// TIA Portal V17 export
// export: Created 2022-07-28T18:02:51.1068585Z, ExportSetting None, DisplayName Totally Integrated Automation Portal, DisplayVersion V17, DisplayName TIA Portal Openness, DisplayVersion V17, DisplayName TIA Portal Teamcenter Gateway, DisplayVersion V17, DisplayName TIA Portal Version Control Interface, DisplayVersion V17, DisplayName TIA Portal Test Suite Advanced, DisplayVersion V17, DisplayName SINAMICS Startdrive Advanced, DisplayVersion V17, DisplayName SINAMICS DCC, DisplayVersion V17, DisplayName SINAMICS Startdrive G130, G150, S120, S150, SINAMICS MV, S210, DisplayVersion V17, DisplayName SINAMICS Startdrive G110M, G120, G120C, G120D, G120P, G115D, DisplayVersion V17, DisplayName STEP 7 Professional, DisplayVersion V17, DisplayName SIMATIC Energy Suite, DisplayVersion V17, DisplayName STEP 7 CFC, DisplayVersion V17, DisplayName STEP 7 Safety, DisplayVersion V17, DisplayName WinCC Advanced / Unified PC, DisplayVersion V17, DisplayName SIMATIC Visualization Architect, DisplayVersion V17
FUNCTION_BLOCK "Lib_FB_SlideGate_Blow"   // FB63, SCL
{ S7_Optimized_Access := 'TRUE' }
// stored: AutoNumber false, MemoryReserve 100, SetENOAutomatically false
   VAR_INPUT
      I_Initialization { ExternalAccessible := 'False'; ExternalVisible := 'False'; ExternalWritable := 'False'} : Bool := FALSE;   // 1 = Restart PLC is active (First scan)
      IR_CycleTime { ExternalAccessible := 'False'; ExternalVisible := 'False'; ExternalWritable := 'False'} : Real := 0.0;   // Time of last PLC cycle, sec
      II_Obj_ID { ExternalAccessible := 'False'; ExternalVisible := 'False'; ExternalWritable := 'False'} : Int := -1;   // Tech ID of object
      I_CmdGeneralReset { ExternalAccessible := 'False'; ExternalVisible := 'False'; ExternalWritable := 'False'} : Bool;   // 0 ⮥ 1 = Input general reset ERROR/Interlocks
      I_One_1s { ExternalAccessible := 'False'; ExternalVisible := 'False'; ExternalWritable := 'False'} : Bool;   // 1 = One cycle per one seccond pulse
      I_EstopHMI { ExternalAccessible := 'False'; ExternalVisible := 'False'; ExternalWritable := 'False'} : Bool := TRUE;   // 0 = HMI/WinCC Emergency stop active
      I_SuppyBox_Ok { ExternalAccessible := 'False'; ExternalVisible := 'False'; ExternalWritable := 'False'} : Bool := TRUE;   // 1 = Release from supply box where exist object
      I_IsOpen { ExternalAccessible := 'False'; ExternalVisible := 'False'; ExternalWritable := 'False'} : Bool;   // Repeat status of opened sensor
      I_IsClose { ExternalAccessible := 'False'; ExternalVisible := 'False'; ExternalWritable := 'False'} : Bool;   // Repeat status of closed sensor
      I_GenFaultMainDrive { ExternalAccessible := 'False'; ExternalVisible := 'False'; ExternalWritable := 'False'} : Bool := TRUE;   // 1 = ППП/Гібридкий контактор/ПЧ в нормі// 0 = Аварія
      I_CmdAutoFromInputFB { ExternalAccessible := 'False'; ExternalVisible := 'False'; ExternalWritable := 'False'} : Bool;   // 1 = Команди AutoMode беруться із входу FB // 0 = Команди AutoMode беруться із масиву AutoArray
      I_CmdAutoOpen { ExternalAccessible := 'False'; ExternalVisible := 'False'; ExternalWritable := 'False'} : Bool;   // (if IB_CmdAutoFromInputFB==1) 1 = In auto mode the motor to run in open direction until the open interlock becomes false, or this input is set low"
      I_CmdAutoClose { ExternalAccessible := 'False'; ExternalVisible := 'False'; ExternalWritable := 'False'} : Bool;   // (if IB_CmdAutoFromInputFB==1) 1 = In auto mode the motor to run in close direction until the close interlock becomes false, or this input is set low"
      I_ManLocalModeActive { ExternalAccessible := 'False'; ExternalVisible := 'False'; ExternalWritable := 'False'} : Bool;   // Switching in external mode ManualLocal if PRM.ManLocalPirority=1(hight)
      I_CmdManLocalOpen { ExternalAccessible := 'False'; ExternalVisible := 'False'; ExternalWritable := 'False'} : Bool;   // 1 = In ManualLocal mode the motor to run in open direction until the open interlock becomes false, or this input is set low
      I_CmdManLocalClose { ExternalAccessible := 'False'; ExternalVisible := 'False'; ExternalWritable := 'False'} : Bool;   // 1 = In ManualLocal mode the motor to run in close direction until the close interlock becomes false, or this input is set low
      IB_InterlocksOpen_8 { ExternalAccessible := 'False'; ExternalVisible := 'False'; ExternalWritable := 'False'} : Byte;   // <>0 = Interlock active - One or more from 8 Interlocks active // 1bit <--> 1 Interlock
      IB_InterlocksClose_8 { ExternalAccessible := 'False'; ExternalVisible := 'False'; ExternalWritable := 'False'} : Byte;   // <>0 = Interlock active - One or more from 8 Interlocks active // 1bit <--> 1 Interlock
      IW_ExternalError_16 { ExternalAccessible := 'False'; ExternalVisible := 'False'; ExternalWritable := 'False'} : Word;   // <>0 = External error active - One or more from 16 error active // 1bit <--> 1 error
      I_ExternalWarning { ExternalAccessible := 'False'; ExternalVisible := 'False'; ExternalWritable := 'False'} : Bool;   // 1 = External Warning
   END_VAR
   VAR_OUTPUT
      Q_CmdOpen { ExternalAccessible := 'False'; ExternalVisible := 'False'; ExternalWritable := 'False'} : Bool;   // 1 = Motor commanded open /Activation output / State transferred to physical output
      Q_IsOpen { ExternalAccessible := 'False'; ExternalVisible := 'False'; ExternalWritable := 'False'} : Bool;   // Repeat status of opened sensor
      Q_IsClose { ExternalAccessible := 'False'; ExternalVisible := 'False'; ExternalWritable := 'False'} : Bool;   // Repeat status of closed sensor
      Q_Reset { ExternalAccessible := 'False'; ExternalVisible := 'False'; ExternalWritable := 'False'} : Bool;   // 1 = Reset faults
      Q_Error { ExternalAccessible := 'False'; ExternalVisible := 'False'; ExternalWritable := 'False'} : Bool;   // This output indicates whether theres an error/fault condition in the motor
      Q_Warning { ExternalAccessible := 'False'; ExternalVisible := 'False'; ExternalWritable := 'False'} : Bool;   // This output indicates whether theres an warning condition in the motor
      Q_Auto { ExternalAccessible := 'False'; ExternalVisible := 'False'; ExternalWritable := 'False'} : Bool;   // 1= Automatic operating mode active
      Q_ManLocal { ExternalAccessible := 'False'; ExternalVisible := 'False'; ExternalWritable := 'False'} : Bool;   // 1= ManualLocal operating mode active
      Q_Stoped { ExternalAccessible := 'False'; ExternalVisible := 'False'; ExternalWritable := 'False'} : Bool;   // 1= Motor Stoped
      Q_Run { ExternalAccessible := 'False'; ExternalVisible := 'False'; ExternalWritable := 'False'} : Bool;   // 1= Motor running
      Q_RunOpen { ExternalAccessible := 'False'; ExternalVisible := 'False'; ExternalWritable := 'False'} : Bool;   // 1= Motor running open
      Q_RunClose { ExternalAccessible := 'False'; ExternalVisible := 'False'; ExternalWritable := 'False'} : Bool;   // 1= Motor running close
      Q_DataErr { ExternalAccessible := 'False'; ExternalVisible := 'False'; ExternalWritable := 'False'} : Bool;   // 1 = Transfer data error occured (ObjDB -> temp, ect)
   END_VAR
   VAR_IN_OUT
      IQ_PLC_CycleInfo : Variant;   // Ref to data about PLC cycle
   END_VAR
   VAR
      s_RequestOpen { ExternalAccessible := 'False'; ExternalVisible := 'False'; ExternalWritable := 'False'} : Bool;   // 1 = Request for start in Open dirrection for all modes
      s_TON_Plausible { ExternalAccessible := 'False'; ExternalVisible := 'False'; ExternalWritable := 'False'} : "Lib_FB_Timer_ON_Simple";
      s_TON_Pause { ExternalAccessible := 'False'; ExternalVisible := 'False'; ExternalWritable := 'False'} : "Lib_FB_Timer_ON_Simple";
      s_TP_Work { ExternalAccessible := 'False'; ExternalVisible := 'False'; ExternalWritable := 'False'} : "Lib_FB_Timer_TP_Simple";
      s_EdgeAuto { ExternalAccessible := 'False'; ExternalVisible := 'False'; ExternalWritable := 'False'} : "Lib_FB_Edge";
      s_EdgeActivOpen { ExternalAccessible := 'False'; ExternalVisible := 'False'; ExternalWritable := 'False'} : "Lib_FB_Edge";
      s_EdgeActivClose { ExternalAccessible := 'False'; ExternalVisible := 'False'; ExternalWritable := 'False'} : "Lib_FB_Edge";
      s_EdgeSim { ExternalAccessible := 'False'; ExternalVisible := 'False'; ExternalWritable := 'False'} : "Lib_FB_Edge";
      s_EdgeLocal { ExternalAccessible := 'False'; ExternalVisible := 'False'; ExternalWritable := 'False'} : "Lib_FB_Edge";
      s_EdgeError { ExternalAccessible := 'False'; ExternalVisible := 'False'; ExternalWritable := 'False'} : "Lib_FB_Edge";
      s_EdgeWarning { ExternalAccessible := 'False'; ExternalVisible := 'False'; ExternalWritable := 'False'} : "Lib_FB_Edge";
   END_VAR
   VAR RETAIN
      s_Simulation { ExternalAccessible := 'False'; ExternalVisible := 'False'; ExternalWritable := 'False'} : Struct   // Data for simulation process
         Obj_DATA_BACKUP : Struct   // MOTOR NORMAL MODE DATA BACKUP FOR SIMULATION MODE
            Config : "_SlideGate_Blow_Config";
            Counters : "_SlideGate_Blow_Counters";
            sud_MotoHours_Electro : "_MotoHours_One";
            sud_MotoHours_Mech : "_MotoHours_One";
         END_STRUCT;
      END_STRUCT;
      s_Obj_Retain_BUp { ExternalAccessible := 'False'; ExternalVisible := 'False'; ExternalWritable := 'False'} : Struct
         Config : "_SlideGate_Blow_Config";
         Counters : "_SlideGate_Blow_Counters";
         Mode : "UDT_Mode";
      END_STRUCT;
   END_VAR
   VAR
      s_TP_ResetOut { ExternalAccessible := 'False'; ExternalVisible := 'False'; ExternalWritable := 'False'} : "Lib_FB_Timer_TP_Simple";
   END_VAR
   VAR_TEMP
      t_DataErr : Bool;   // 1 = Transfer data error occured (ObjDB -> temp, ect)
      t_PlausibleCondition : Bool;   // 1 = Conition for detect plausible error
      t_ReleaseStart : Bool;   // 1 = Release for start in any mode
      t_RequestActive : Bool;   // 1 = Request is active for any mode in any dirrection
      t_RequestOpenActive : Bool;   // 1 = Request is active for any mode in Open dirrection
      t_RequestCloseActive : Bool;   // 1 = Request is active for any mode in Close dirrection
      t_ResetLogic : Bool;   // 1 = Reset all signals for logic
      ti_CMDLogic : Int;   // Command word for logic
      tui_NumObjDB : UInt;   // Number of DB for storage object data
      tui_MaxObjects : UInt;   // Max number of objects in plant
      tui_DB_ShiftHMI : UInt;   // Object DB number shift
      tui_DB_ShiftPLC : UInt;   // Object DB number shift
      tui_DBSens_ShiftHMI : UInt;   // Object DB number shift
      tui_DBSens_ShiftPLC : UInt;   // Object DB number shift
      t_ObjAny_HMI : DB_ANY;   // Ref to object data
      t_ObjVar_HMI : Variant;   // Ref to object data
      t_ObjAny_PLC : DB_ANY;   // Ref to object data
      t_ObjVar_PLC : Variant;   // Ref to object data
      t_PB_HMI : Struct   // Buttons from HMI
         ResetError : Bool;   // + set-->CMD_ALMACK_tag -Reset errors pushbutton
         ManRunOpen : Bool;   // - Move Open in manual mode pushbutton
         ManRunClose : Bool;   // - Move Close in manual mode pushbutton
         ResetGeneralReset : Bool;   // -Reset Error + Interlock
         CntResetALL : Bool;   // - обнулити всі лічильники - (Total+Last+Alm+Wrn+)
         CntResetTimeTOT : Bool;   // - обнулити лічильник мотогодин (Total+Last)
         CntResetActTOT : Bool;   // - обнулити запусків (Total+Last)
         spare7 : Bool;
         spare8 : Bool;
         spare9 : Bool;
         spare10 : Bool;
         spare11 : Bool;
         spare12 : Bool;
         spare13 : Bool;
         spare14 : Bool;
         spare15 : Bool;
         spare16 : Bool;
         spare17 : Bool;
         spare18 : Bool;
         spare19 : Bool;
         spare20 : Bool;
         spare21 : Bool;
         spare22 : Bool;
         spare23 : Bool;
         spare24 : Bool;
         spare25 : Bool;
         spare26 : Bool;
         spare27 : Bool;
         spare28 : Bool;
         spare29 : Bool;
         spare30 : Bool;
         spare31 : Bool;
      END_STRUCT;
      t_Obj_HMI : "Lib_UDT_SlideGate_Blow_HMI";   // Object data
      t_Obj_PLC : "Lib_UDT_SlideGate_Blow_PLC";
      t_PLC_CycleInfo : "Lib_PLC_CycleInfo";   // Data about PLC cycle
      t_AutoControl : "Lib_UDT_AutoControl";   // Data for auto control module for current element
      t_InternalData : "Lib_UDT_Int";   // Internal data
      t_AutoControl_CMD : Struct   // Commands from auto control module for current element
         CmdAutoOpen : Bool;
         CmdAutoClose : Bool;
         CmdAutoOpenRaw : Bool;
         CmdAutoCloseRaw : Bool;
      END_STRUCT;
      t_Buffer : Array[0..100] of Byte;   // Buffer for use serialize
   END_VAR
   VAR CONSTANT
      cr_TimePlausible : Real := 5.0;   // Time for detectplausible error, s
      cr_TimeAddWalkErr : Real := 20.0;   // Additional time for walk error after autocalibrate, %
   END_VAR
BEGIN

   REGION Initialization/read data from out DB
       //Set internal data
       "Lib_FC_GenMoto_InitInternal"(#t_InternalData);

       //Reinit gen data
       #t_DataErr := false;
       #t_Obj_HMI.Config.w_enableExternalErrors_16 := w#16#FFFF;
       #t_Obj_HMI.Config.b_bypassInterlocksForward_8 := b#16#ff;
       #t_Obj_HMI.Config.b_bypassInterlocksReverse_8 := b#16#ff;
       #tui_MaxObjects := "D_General_ProgramDATA".ui_MaxObjects;
       #tui_DB_ShiftHMI := "D_General_ProgramDATA".ui_Shift_DB_HMI;
       #tui_DB_ShiftPLC := "D_General_ProgramDATA".ui_Shift_DB_PLC;
       #tui_DBSens_ShiftHMI := "D_General_ProgramDATA".ui_Shift_DBSens_HMI;
       #tui_DBSens_ShiftPLC := "D_General_ProgramDATA".ui_Shift_DBSens_PLC;
       //Read data PLC
       VariantGet(SRC := #IQ_PLC_CycleInfo,
                  DST => #t_PLC_CycleInfo);

       //Read Object data
       //Reinit temp values
       #t_Obj_HMI := "D_ZeroTypes".SlideGate_Blow_HMI;
       #t_Obj_PLC := "D_ZeroTypes".SlideGate_Blow_PLC;

       IF #II_Obj_ID >= 0
       THEN
           //Read HMI data
           #tui_NumObjDB := INT_TO_UINT(#II_Obj_ID) + #tui_DB_ShiftHMI;
           #t_ObjAny_HMI := UINT_TO_DB_ANY(#tui_NumObjDB);
           #t_ObjVar_HMI := DB_ANY_TO_VARIANT(in := #t_ObjAny_HMI, err => #t_InternalData.i_Tmp);

           //If DB exist and convertion without error
           IF #t_InternalData.i_Tmp = 0
           THEN
               VariantGet(SRC := #t_ObjVar_HMI,
                          DST => #t_Obj_HMI);
           ELSE
               #t_DataErr := true;
           END_IF;

           //Read PLC data
           #tui_NumObjDB := INT_TO_UINT(#II_Obj_ID) + #tui_DB_ShiftPLC;
           #t_ObjAny_PLC := UINT_TO_DB_ANY(#tui_NumObjDB);
           #t_ObjVar_PLC := DB_ANY_TO_VARIANT(in := #t_ObjAny_PLC, err => #t_InternalData.i_Tmp);

           //If DB exist and convertion without error
           IF #t_InternalData.i_Tmp = 0
           THEN
               VariantGet(SRC := #t_ObjVar_PLC,
                          DST => #t_Obj_PLC);
           ELSE
               #t_DataErr := true;
           END_IF;

       ELSE
           #t_DataErr := true;
       END_IF;

       //Read general info data
       #t_AutoControl := "DB_AutoControl_arr".AutoControl_arr[#tui_MaxObjects];
       CASE #II_Obj_ID OF
           0..999:  // ID of element in range
               #t_AutoControl := "DB_AutoControl_arr".AutoControl_arr[#II_Obj_ID];
           ELSE
               ;
       END_CASE;

       //Read retain data if initialization is active
       IF #I_Initialization
       THEN
           #t_Obj_HMI.Config := #s_Obj_Retain_BUp.Config;
           #t_Obj_HMI.Counters := #s_Obj_Retain_BUp.Counters;
           #t_Obj_PLC.Mode := #s_Obj_Retain_BUp.Mode;
       END_IF;
   END_REGION
   //---------------------------------------------------------------
   //---------------------------------------------------------------
   REGION Define CMD for block logic 
       //Reinit logic CMD
       #ti_CMDLogic := 0;

       //Define CMD by priority modes
       "Lib_FC_GenMoto_ChoiceCMD"(I_Mode := #t_Obj_PLC.Mode,
                                  QI_CMD_Logic => #ti_CMDLogic,
                                  IQI_CMD_Global := #t_PLC_CycleInfo.CMD_GLOBAL,
                                  IQI_CMD_Auto := #t_AutoControl.Global_CMD,
                                  IQI_CMD_HMI := #t_Obj_HMI.i_CMD);
   END_REGION
   //---------------------------------------------------------------
   //---------------------------------------------------------------
   REGION Switch modes  
       "Lib_FC_GenMoto_SwitchMode"(I_ManLocalModeActive := #I_ManLocalModeActive,
                                   IQI_CMD_Logic := #ti_CMDLogic,
                                   IQ_Mode := #t_Obj_PLC.Mode,
                                   IQ_ObjDataConfig := #t_Obj_HMI.Config,
                                   IQ_BUpDataConfig := #s_Simulation.Obj_DATA_BACKUP.Config,
                                   IQ_ObjDataCounters := #t_Obj_HMI.Counters,
                                   IQ_BUpDataCounters := #s_Simulation.Obj_DATA_BACKUP.Counters);

       #s_EdgeAuto(IB_Initialisation:=#I_Initialization,
                   IB_Input:=#t_Obj_PLC.Mode.Auto);
       #s_EdgeSim(IB_Initialisation:=#I_Initialization,
                  IB_Input:=#t_Obj_PLC.Mode.Simulation);
       #s_EdgeLocal(IB_Initialisation:=#I_Initialization,
                    IB_Input:=#t_Obj_PLC.Mode.ManualLocal);

   END_REGION
   //---------------------------------------------------------------
   //---------------------------------------------------------------
   REGION Commands & release for start in auto mode
       //Raw command for start in auto mode
       //-------------------------------------
       IF #I_CmdAutoFromInputFB
       THEN // Auto CMD from FB INPUT
           #t_AutoControl_CMD.CmdAutoOpenRaw := #I_CmdAutoOpen
           AND #t_Obj_PLC.Mode.Auto;
           #t_AutoControl_CMD.CmdAutoCloseRaw := #I_CmdAutoClose
           AND #t_Obj_PLC.Mode.Auto;

       ELSE // Auto CMD from AutoControl_array DB

           IF #t_Obj_PLC.Mode.Auto
           THEN
               IF #s_TP_Work.QB_TimerOut
               THEN
                   #t_AutoControl.CTW.%W0 := W#16#1;
                   #t_AutoControl.StatusGen.Release := true;
               ELSE
                   #t_AutoControl.CTW.%W0 := W#16#0;
                   #t_AutoControl.StatusGen.Release := false;
               END_IF;
           ELSE
               #t_AutoControl.CTW := dW#16#0;
               #t_AutoControl.StatusGen.Release := false;
           END_IF;

           #t_AutoControl_CMD.CmdAutoOpenRaw := (WORD_TO_UINT(#t_AutoControl.CTW.%W0) > 0)
           AND #t_AutoControl.StatusGen.Release;
           #t_AutoControl_CMD.CmdAutoCloseRaw := (WORD_TO_UINT(#t_AutoControl.CTW.%W1) > 0)
           AND #t_AutoControl.StatusGen.Release;

       END_IF;
       //-------------------------------------
       //-------------------------------------
       //Processed auto mode commands
       #t_AutoControl_CMD.CmdAutoOpen := #t_AutoControl_CMD.CmdAutoOpenRaw;
       #t_AutoControl_CMD.CmdAutoClose := #t_AutoControl_CMD.CmdAutoCloseRaw;

       REGION Timers for work and pause 
           #s_TON_Pause(IR_CycleTime:=#IR_CycleTime,
                        IB_StartTimerInput:=NOT #s_TP_Work.QB_TimerOut,
                        IB_ResetTimer:=NOT #t_Obj_PLC.Mode.Auto
                        OR NOT #t_Obj_PLC.State.Ready,
                        IR_SpTime:=#t_Obj_HMI.Config.r_SP_TimePause);

           #s_TP_Work(IR_CycleTime:=#IR_CycleTime,
                      IB_StartTimerInput:=#s_TON_Pause.QB_TimerOut
                      OR #s_EdgeAuto.QB_EdgePos,
                      IB_ResetTimer:=NOT #t_Obj_PLC.Mode.Auto
                      OR NOT #t_Obj_PLC.State.Ready,
                      IR_SpTime:=#t_Obj_HMI.Config.r_SP_TimeWork);

           //Left time
           IF #t_Obj_PLC.Mode.Auto
           THEN
               IF #s_TON_Pause.sR_Cv_ToDone > 0.0
               THEN
                   #t_Obj_HMI.Config.r_PV_LeftTime := #s_TON_Pause.sR_Cv_ToDone;
               ELSE
                   #t_Obj_HMI.Config.r_PV_LeftTime := 0.0;
               END_IF;
           ELSE
               #t_Obj_HMI.Config.r_PV_LeftTime := 0.0;
           END_IF;
       END_REGION


       //Reset release bit
      // #t_AutoControl.StatusGen.Release := false; 
   END_REGION
   //---------------------------------------------------------------
   //---------------------------------------------------------------
   REGION Convert commands to bit
       //Reinit all bits
       SCATTER(IN := #t_InternalData.d_Alw0,
               OUT => #t_PB_HMI);

       //Read commands and set apropriate bits
       CASE #ti_CMDLogic OF
           12:  // Start open in manual mode
               #t_PB_HMI.ManRunOpen := true;
           13:  // Start close in manual mode
               #t_PB_HMI.ManRunClose := true;
           19: //Start autocalibrate process
               #t_Obj_HMI.Config.b.SimAutoSensorChange := true;
           20: //Enable/disable auto change of sensor state in simulation mode
               #t_Obj_HMI.Config.b.bit_3 := NOT #t_Obj_HMI.Config.b.bit_3;
           31:  // Reset general (faults and interlocks)
               #t_PB_HMI.ResetGeneralReset := true;
           32: // Reset errors
               #t_PB_HMI.ResetError := true;
           40: //Reset all counters
               #t_PB_HMI.CntResetALL := true;
           41: //Reset counters of motohours
               #t_PB_HMI.CntResetTimeTOT := true;
           42: //Reset counters of starts
               #t_PB_HMI.CntResetActTOT := true;
           ELSE
               ;
       END_CASE;

       //General bits for logic
       //General reset
       #t_ResetLogic := #t_PB_HMI.ResetError
       OR #t_PB_HMI.ResetGeneralReset
       OR #I_CmdGeneralReset;

       //Reset for out of block
       #s_TP_ResetOut(IR_CycleTime := #IR_CycleTime,
                      IB_StartTimerInput := #t_ResetLogic,
                      IR_SpTime := 1.5);
   END_REGION
   //---------------------------------------------------------------
   //---------------------------------------------------------------
   REGION Process switch inputs(isOpen/isClose)
       //For not simulation mode
       IF NOT #t_Obj_PLC.Mode.Simulation
       THEN
           #t_Obj_PLC.State.Opened := #I_IsOpen;
           #t_Obj_PLC.State.Closed := #I_IsClose;
       ELSE //For simulation mode

           //If not active autochange sensor state
           IF NOT #t_Obj_HMI.Config.b.SimAutoSensorChange
           THEN
               CASE #ti_CMDLogic OF
                   114: //Change opened input
                       #t_Obj_PLC.State.Opened := NOT #t_Obj_PLC.State.Opened;
                   115: //Change closed input
                       #t_Obj_PLC.State.Closed := NOT #t_Obj_PLC.State.Closed;
                   ELSE
                       ;
               END_CASE;
           ELSE
               IF #s_RequestOpen
               THEN
                   #t_Obj_PLC.State.Opened := true;
                   #t_Obj_PLC.State.Closed := false;
               END_IF;
               IF NOT #s_RequestOpen
               THEN
                   #t_Obj_PLC.State.Opened := false;
                   #t_Obj_PLC.State.Closed := true;
               END_IF;
           END_IF;
       END_IF;

   END_REGION
   //---------------------------------------------------------------
   //---------------------------------------------------------------
   REGION Proccess faults, warnings, interlocks and status bits

       REGION Reinit words
           // Reinit alarm words
           IF #t_ResetLogic
               OR #I_Initialization
               OR #t_Obj_PLC.Mode.Disable
               OR #t_Obj_PLC.Mode.Repair
           THEN
               #t_Obj_HMI.Status.w_ALW1 := #t_InternalData.w_Alw0;
               #t_Obj_HMI.Status.w_ALW2 := #t_InternalData.w_Alw0;
               #t_Obj_HMI.Status.w_ALW3 := #t_InternalData.w_Alw0;
               #t_Obj_HMI.Status.w_ALW4 := #t_InternalData.w_Alw0;
               #t_Obj_HMI.Status.w_ALW5 := #t_InternalData.w_Alw0;
               //#t_Obj_PLC.State := "DB_ZeroTypes".Shutter_Gen_PLC.State;
               #t_Obj_PLC.Alarm := "D_ZeroTypes".SlideGate_Blow_PLC.Alarm;
           END_IF;

           //Reinit STW words
           #t_Obj_HMI.Status.dw_STW_1 := #t_InternalData.d_Alw0;
           #t_Obj_HMI.Status.dw_STW_2 := #t_InternalData.d_Alw0;
           #t_Obj_HMI.Status.dw_STW := #t_InternalData.d_Alw0;

           //Reinit interlocks words
           #t_Obj_HMI.Status.dw_ILW_Open := #t_InternalData.d_Alw0;
           #t_Obj_HMI.Status.dw_ILW_Close := #t_InternalData.d_Alw0;
       END_REGION

       //Interlocks
       #t_Obj_PLC.Alarm.InterlockOpen := ((#t_Obj_HMI.Config.b_bypassInterlocksForward_8
       AND #IB_InterlocksOpen_8) <> b#16#0)
       AND NOT #t_Obj_PLC.Mode.Disable
       AND NOT #t_Obj_PLC.Mode.Service;

       #t_Obj_PLC.Alarm.InterlockClose := ((#t_Obj_HMI.Config.b_bypassInterlocksReverse_8
       AND #IB_InterlocksClose_8) <> b#16#0)
       AND NOT #t_Obj_PLC.Mode.Disable
       AND NOT #t_Obj_PLC.Mode.Service;

       #t_Obj_HMI.Status.dw_ILW_Open.%B0 := #IB_InterlocksOpen_8;
       #t_Obj_HMI.Status.dw_ILW_Close.%B0 := #IB_InterlocksClose_8;

       REGION Faults common for sim and gen modes
           IF NOT #t_Obj_PLC.Mode.Disable
           THEN
               //Emergency stop from HMI 
               #t_Obj_PLC.Alarm.EstopHMI := NOT #I_EstopHMI;

               //External warning
               #t_Obj_PLC.Alarm.ExtWarning := #I_ExternalWarning;

               //External error
               #t_Obj_HMI.Status.dw_EEW.%W0 := #IW_ExternalError_16;
               #t_Obj_PLC.Alarm.ExtError := (#IW_ExternalError_16
               AND #t_Obj_HMI.Config.w_enableExternalErrors_16) <> w#16#0;

               //Internal warning
               #t_Obj_PLC.Alarm.IntWarning := #t_Obj_PLC.Alarm.UndefPosition;

               //Fault of supply box
               #t_Obj_PLC.Alarm.FaultSupplyBox := NOT #I_SuppyBox_Ok;

               //Both request
               #t_Obj_PLC.Alarm.BothCommandToStart := false;

               //Sensor error 
               #t_Obj_PLC.Alarm.SensorError := false;

               //Error plausible (booth sensors, open when close active ect.)
               //Time befor plausible error detect
               #t_Obj_PLC.Alarm.ErrPlausible := #s_TON_Plausible.QB_TimerOut
               OR (#t_Obj_PLC.Alarm.ErrPlausible
               AND NOT #t_ResetLogic)
               AND NOT #I_Initialization;

               //Undefined position
               #t_Obj_PLC.Alarm.UndefPosition := false;
           END_IF;

       END_REGION

       REGION Faults different for sim and gen modes
           IF NOT #t_Obj_PLC.Mode.Simulation 
               AND NOT #t_Obj_PLC.Mode.Disable
           THEN
               //General fault of main drive (soft starter ect)
               #t_Obj_PLC.Alarm.TripGenMainDrive := (NOT #I_GenFaultMainDrive
               OR (NOT #t_ResetLogic
               AND #t_Obj_PLC.Alarm.TripGenMainDrive))
               AND NOT #I_Initialization;

           ELSIF #t_Obj_PLC.Mode.Simulation
               AND NOT #t_Obj_PLC.Mode.Disable
           THEN

               CASE #ti_CMDLogic OF
                   110:  //General fault of main drive
                       #t_Obj_PLC.Alarm.TripGenMainDrive := NOT #t_Obj_PLC.Alarm.TripGenMainDrive;
                   113:  //Both commands to motor is active
                       #t_Obj_PLC.Alarm.BothCommandToStart := NOT #t_Obj_PLC.Alarm.BothCommandToStart;
                   120: //Plausible error
                       #t_Obj_PLC.Alarm.ErrPlausible := NOT #t_Obj_PLC.Alarm.ErrPlausible;
                   ELSE
                       ;
               END_CASE;

           END_IF;

           REGION Timers, edges ect.

                   //Plausible error
                   #t_PlausibleCondition := false;

                   #s_TON_Plausible(IR_CycleTime := #IR_CycleTime,
                                    IB_StartTimerInput := #t_PlausibleCondition
                                    AND NOT #t_Obj_PLC.Alarm.ErrPlausible,
                                    IB_ResetTimer := #t_Obj_PLC.Mode.Disable
                                    OR #t_Obj_PLC.Mode.Service
                                    OR #t_ResetLogic
                                    OR #I_Initialization
                                    OR #t_PlausibleCondition,
                                    IR_SpTime := #cr_TimePlausible);

           END_REGION
       END_REGION

       REGION Some faults is active

           #t_Obj_PLC.State.Error := #t_Obj_PLC.Alarm.SensorError
           OR #t_Obj_PLC.Alarm.EstopHMI
           OR #t_Obj_PLC.Alarm.ExtError
           OR #t_Obj_PLC.Alarm.FaultSupplyBox
           OR #t_Obj_PLC.Alarm.BothCommandToStart
           OR #t_Obj_PLC.Alarm.ErrPlausible
           OR #t_Obj_PLC.Alarm.TripGenMainDrive
           ;

       END_REGION
   END_REGION
   //---------------------------------------------------------------
   //---------------------------------------------------------------
   REGION Release for start in any mode
       #t_ReleaseStart := NOT #t_Obj_PLC.State.Error
       AND NOT #t_Obj_PLC.Mode.Disable
       AND NOT #t_Obj_PLC.Mode.Repair
       AND NOT #s_EdgeAuto.QB_EdgeNeg
       AND NOT #s_EdgeSim.QB_EdgeNeg
       AND NOT #s_EdgeLocal.QB_EdgeNeg
       AND NOT #I_Initialization;
   END_REGION
   //---------------------------------------------------------------
   //---------------------------------------------------------------
   REGION Requests for start in any dirrections

       REGION Request in open dirrection
           //Release for start
           #s_RequestOpen := #t_ReleaseStart
           AND NOT #t_Obj_PLC.Alarm.InterlockOpen

           //Start command in auto mode
           AND ((#t_Obj_PLC.Mode.Auto
           AND #t_AutoControl_CMD.CmdAutoOpen)

           //Start in manual remote mode
           OR ((#t_Obj_PLC.Mode.ManualRemote
           OR #t_Obj_PLC.Mode.Service)
           AND (#t_PB_HMI.ManRunOpen
           OR #s_RequestOpen)
           AND NOT #t_PB_HMI.ManRunClose)

           //Start in manual local mode
           OR (#t_Obj_PLC.Mode.ManualLocal
           AND #I_CmdManLocalOpen)
           );
       END_REGION
   END_REGION
   //---------------------------------------------------------------
   //---------------------------------------------------------------
   REGION Call block of motor 
       REGION Pulses for motor running
           #s_EdgeActivOpen(IB_Initialisation := #I_Initialization,
                            IB_Input := #s_RequestOpen
           );
           #s_EdgeActivClose(IB_Initialisation := #I_Initialization,
                             IB_Input := NOT #s_RequestOpen
           );
       END_REGION
   END_REGION

   REGION General states
       IF NOT #t_Obj_PLC.Mode.Disable
           AND NOT #t_Obj_PLC.Mode.Repair
       THEN
           //General states 
           #t_Obj_PLC.Alarm.InCmdAutoOpen := #t_AutoControl_CMD.CmdAutoOpen;
           #t_Obj_PLC.Alarm.InCmdAutoClose := #t_AutoControl_CMD.CmdAutoClose;
           #t_Obj_PLC.Alarm.SigOutOpening := #Q_CmdOpen;
           #t_Obj_PLC.Alarm.SigOutClosing := NOT #Q_CmdOpen;
           #t_Obj_PLC.Alarm.RequestForward  := #s_RequestOpen;
           #t_Obj_PLC.Alarm.RequestReverse  := NOT #s_RequestOpen;
           #t_Obj_PLC.Alarm.RunOpen := #s_RequestOpen;
           #t_Obj_PLC.Alarm.RunClose := NOT #s_RequestOpen;
           #t_Obj_PLC.Alarm.Closed := #t_Obj_PLC.State.Closed;
           #t_Obj_PLC.Alarm.Opened := #t_Obj_PLC.State.Opened;
           #t_Obj_PLC.Alarm.AW4_bit_3 := #t_Obj_HMI.Config.b.SimAutoSensorChange;
           #t_Obj_PLC.Alarm.SimAutochangeActive := #t_Obj_HMI.Config.b.bit_3;

           #t_Obj_PLC.State.Warning := #I_ExternalWarning
           OR  #t_Obj_PLC.Alarm.IntWarning;
           #t_Obj_PLC.State.Maintenance := #t_Obj_PLC.Alarm.MaintenanceElectroServ
           OR #t_Obj_PLC.Alarm.MaintenanceMechanoServ;
           #t_Obj_PLC.State.Interlocked := #t_Obj_PLC.Alarm.InterlockOpen
           OR #t_Obj_PLC.Alarm.InterlockClose;
           #t_Obj_PLC.State.Ready := #t_ReleaseStart;
           #t_Obj_PLC.State.Stoped := NOT #s_RequestOpen;
           #t_Obj_PLC.State.Run := true;
           #t_Obj_PLC.State.RunOpen := #s_RequestOpen;
           #t_Obj_PLC.State.RunClose := NOT #s_RequestOpen;
           #t_Obj_PLC.State.ActiveH := false;
           #t_Obj_PLC.State.ActiveL := false;
       END_IF;

       //States for all modes
       #t_Obj_PLC.Alarm.Disable  := #t_Obj_PLC.Mode.Disable;
       #t_Obj_PLC.Alarm.ManualRemote  := #t_Obj_PLC.Mode.ManualRemote;
       #t_Obj_PLC.Alarm.Auto  := #t_Obj_PLC.Mode.Auto;
       #t_Obj_PLC.Alarm.ManualLocal  := #t_Obj_PLC.Mode.ManualLocal;
       #t_Obj_PLC.Alarm.Service  := #t_Obj_PLC.Mode.Service;
       #t_Obj_PLC.Alarm.RepairOn  := #t_Obj_PLC.Mode.Repair;
       #t_Obj_PLC.Alarm.IndependentOn := #t_Obj_PLC.Mode.Independent;
       #t_Obj_PLC.Alarm.SimulationOn  := #t_Obj_PLC.Mode.Simulation;
       #t_Obj_PLC.Alarm.RepairOff  := NOT #t_Obj_PLC.Mode.Repair;
       #t_Obj_PLC.Alarm.IndependentOff  := NOT #t_Obj_PLC.Mode.Independent;
       #t_Obj_PLC.Alarm.SimulationOff  := NOT #t_Obj_PLC.Mode.Simulation;
       #t_Obj_PLC.Alarm.Stopped  := false;

       REGION Pulses for new states
           #s_EdgeError(IB_Initialisation := #I_Initialization,
                      IB_Input := #t_Obj_PLC.State.Error);
           #s_EdgeWarning(IB_Initialisation := #I_Initialization,
                        IB_Input := #t_Obj_PLC.State.Warning);
       END_REGION
   END_REGION
   //---------------------------------------------------------------
   //---------------------------------------------------------------
   REGION Counters
   //Maintenance counters
   "Lib_FC_General_CountMotoHours"(II_Obj_ID := #II_Obj_ID,
                                   I_One_1s := #I_One_1s,
                                   I_Run := #s_RequestOpen,
                                   I_PosPulseSimMode := #s_EdgeSim.QB_EdgePos,
                                   I_NegPulseSimMode := #s_EdgeSim.QB_EdgeNeg,
                                   Q_MaintenanceElectroServ => #t_Obj_PLC.Alarm.MaintenanceElectroServ,
                                   Q_MaintenanceMechanoServ => #t_Obj_PLC.Alarm.MaintenanceMechanoServ,
                                   IQUD_BacUpElectro := #s_Simulation.Obj_DATA_BACKUP.sud_MotoHours_Electro,
                                   IQUD_BacUpMechanic := #s_Simulation.Obj_DATA_BACKUP.sud_MotoHours_Mech);

   //Total operating time
   IF (#s_RequestOpen)
       AND #I_One_1s
   THEN
       #t_Obj_HMI.Counters.di_TimeOper_Tot += 1;
   END_IF;

   //Counter starts
   IF  ((#s_EdgeActivOpen.QB_EdgePos))
   THEN
       #t_Obj_HMI.Counters.di_Activ_tot += 1;
   END_IF;

   //Reset general counters
   IF #t_PB_HMI.CntResetALL
   THEN
       #t_Obj_HMI.Counters.di_TimeOper_Tot := 0;
       #t_Obj_HMI.Counters.di_Activ_tot := 0;
   END_IF;

   IF #t_PB_HMI.CntResetTimeTOT
   THEN
       #t_Obj_HMI.Counters.di_TimeOper_Tot := 0;
   END_IF;

   IF #t_PB_HMI.CntResetActTOT
   THEN
       #t_Obj_HMI.Counters.di_Activ_tot := 0;
   END_IF;


   END_REGION
   //---------------------------------------------------------------
   //---------------------------------------------------------------
   REGION PLC states
       "Lib_FC_Mot_CycleInfo_Count_State"(Alarm := #t_Obj_PLC.State.Error,
                                          AlarmNew := #s_EdgeError.QB_EdgePos,
                                          Warning := #t_Obj_PLC.State.Warning,
                                          WarningNew := #s_EdgeWarning.QB_EdgePos,
                                          Estop := #t_Obj_PLC.Alarm.AW1_bit_0
                                          OR #t_Obj_PLC.Alarm.EstopHMI,
                                          Interlocked := #t_Obj_PLC.State.Interlocked,
                                          InterlockBypassed := false,
                                          Manual := #t_Obj_PLC.Mode.ManualRemote
                                          OR #t_Obj_PLC.Mode.ManualLocal,
                                          Simulation := #t_Obj_PLC.Mode.Simulation,
                                          Error_PSL := NOT #I_SuppyBox_Ok,
                                          PLC_CycleInfo := #t_PLC_CycleInfo);

   END_REGION
   //---------------------------------------------------------------
   //---------------------------------------------------------------
   REGION Write STW and Alarm bits into words

       //Wrapping Alarm bits in words
       #t_InternalData.di_Tmp := 0;
       #t_InternalData.i_Tmp := Serialize(SRC_VARIABLE := #t_Obj_PLC.Alarm, DEST_ARRAY => #t_Buffer, POS := #t_InternalData.di_Tmp);
       #t_Obj_HMI.Status.w_ALW1.%B0 := #t_Buffer[0];
       #t_Obj_HMI.Status.w_ALW1.%B1 := #t_Buffer[1];
       #t_Obj_HMI.Status.w_ALW2.%B0 := #t_Buffer[2];
       #t_Obj_HMI.Status.w_ALW2.%B1 := #t_Buffer[3];
       #t_Obj_HMI.Status.w_ALW3.%B0 := #t_Buffer[4];
       #t_Obj_HMI.Status.w_ALW3.%B1 := #t_Buffer[5];
       #t_Obj_HMI.Status.w_ALW4.%B0 := #t_Buffer[6];
       #t_Obj_HMI.Status.w_ALW4.%B1 := #t_Buffer[7];
       #t_Obj_HMI.Status.w_ALW5.%B0 := #t_Buffer[8];
       #t_Obj_HMI.Status.w_ALW5.%B1 := #t_Buffer[9];

       //Wrapping STW bits
       //States
       #t_InternalData.di_Tmp := 0;
       #t_InternalData.i_Tmp := Serialize(SRC_VARIABLE := #t_Obj_PLC.State, DEST_ARRAY => #t_Buffer, POS := #t_InternalData.di_Tmp);

       //Modes
       #t_InternalData.di_Tmp := 2;
       #t_InternalData.i_Tmp := Serialize(SRC_VARIABLE := #t_Obj_PLC.Mode, DEST_ARRAY => #t_Buffer, POS := #t_InternalData.di_Tmp);

       #t_Obj_HMI.Status.dw_STW.%B0 := #t_Buffer[0]; //States W1
       #t_Obj_HMI.Status.dw_STW.%B1 := #t_Buffer[1]; //States W2
       #t_Obj_HMI.Status.dw_STW.%B2 := #t_Buffer[2]; //Modes W1
       #t_Obj_HMI.Status.dw_STW.%B3 := #t_Buffer[3]; //Modes W2

   END_REGION
   //---------------------------------------------------------------
   //---------------------------------------------------------------
   REGION Write data to HMI and BUp storage
       //HMI data
       #t_Obj_HMI.i_ID := #II_Obj_ID;
       #t_Obj_HMI.i_CLSID := 63;

       //BUp retain data
       //Read retain data if initialization is active
       IF NOT #I_Initialization
       THEN
           #s_Obj_Retain_BUp.Config := #t_Obj_HMI.Config;
           #s_Obj_Retain_BUp.Counters := #t_Obj_HMI.Counters;
           #s_Obj_Retain_BUp.Mode := #t_Obj_PLC.Mode;
       END_IF;
   END_REGION
   //---------------------------------------------------------------
   //---------------------------------------------------------------
   REGION Wrap data for automode module
       #t_AutoControl.STW_HMI := #t_InternalData.d_Alw0;
       #t_AutoControl.STW := #t_InternalData.d_Alw0;

       #t_AutoControl.Mode := #t_Obj_PLC.Mode;
       #t_AutoControl.CLSID := #t_Obj_HMI.i_CLSID;
       #t_AutoControl.StatusGen.Fault := #t_Obj_PLC.State.Error;
       #t_AutoControl.StatusGen.Ready := #t_Obj_PLC.State.Ready;
       #t_AutoControl.StatusGen.ControlAchieve := (#t_AutoControl_CMD.CmdAutoOpen
       AND #t_Obj_PLC.State.Opened)
       OR (#t_AutoControl_CMD.CmdAutoClose
       AND #t_Obj_PLC.State.Closed);

       #t_InternalData.di_Tmp := 0;
       #t_InternalData.i_Tmp := Serialize(SRC_VARIABLE := #t_AutoControl.StatusGen, DEST_ARRAY => #t_Buffer, POS := #t_InternalData.di_Tmp);
       #t_InternalData.di_Tmp := 2;
       #t_InternalData.i_Tmp := Serialize(SRC_VARIABLE := #t_AutoControl.Mode, DEST_ARRAY => #t_Buffer, POS := #t_InternalData.di_Tmp);

       #t_AutoControl.STW_HMI.%B0 := #t_Buffer[0];
       #t_AutoControl.STW_HMI.%B1 := #t_Buffer[1];
       #t_AutoControl.STW_HMI.%B2 := #t_Buffer[2];
       #t_AutoControl.STW_HMI.%B3 := #t_Buffer[3];
       #t_AutoControl.STW_HMI.%X16 := false;

       IF #t_AutoControl_CMD.CmdAutoOpen
           AND #t_Obj_PLC.State.Opened
       THEN
           #t_AutoControl.STW.%W0 := #t_AutoControl.CTW.%W0;
       END_IF;

       IF #t_AutoControl_CMD.CmdAutoClose
           AND #t_Obj_PLC.State.Closed
       THEN
           #t_AutoControl.STW.%W1 := #t_AutoControl.CTW.%W1;
       END_IF;
   END_REGION
   //---------------------------------------------------------------
   //---------------------------------------------------------------
   REGION Write data to out DB
       //Write data  PLC
       VariantPut(SRC := #t_PLC_CycleInfo,
                  DST := #IQ_PLC_CycleInfo);

       //Write Object data
       //DB num 
       IF #II_Obj_ID >= 0
           AND NOT #t_DataErr
       THEN
           //Write HMI data
           VariantPut(SRC := #t_Obj_HMI,
                      DST := #t_ObjVar_HMI);

           //Write PLC data
           VariantPut(SRC := #t_Obj_PLC,
                      DST := #t_ObjVar_PLC);
       ELSE
           #t_DataErr := true;
       END_IF;

       //Write general info data
       CASE #II_Obj_ID OF
           0..999:  // ID of element in range
               "DB_AutoControl_arr".AutoControl_arr[#II_Obj_ID] := #t_AutoControl;
           ELSE
               ;
       END_CASE;
   END_REGION
   //---------------------------------------------------------------
   //---------------------------------------------------------------
   REGION Outputs of block
       #Q_CmdOpen := #s_RequestOpen;
       #Q_IsOpen := #t_Obj_PLC.State.Opened;
       #Q_IsClose := #t_Obj_PLC.State.Closed;
       #Q_Reset := #s_TP_ResetOut.QB_TimerOut;
       #Q_Error := #t_Obj_PLC.State.Error;
       #Q_Warning := #t_Obj_PLC.State.Warning;
       #Q_Auto := #t_Obj_PLC.Mode.Auto;
       #Q_ManLocal := #t_Obj_PLC.Mode.ManualLocal;
       #Q_Stoped := #t_Obj_PLC.State.Stoped;
       #Q_Run := #t_Obj_PLC.State.Run;
       #Q_RunOpen := #t_Obj_PLC.State.RunOpen;
       #Q_RunClose := #t_Obj_PLC.State.RunClose;
       #Q_DataErr := #t_DataErr;
   END_REGION

   //Test text 21.02.2022 zzz
END_FUNCTION_BLOCK
